// TIA Portal V16 export
// export: Created 2022-03-04T10:51:32.4810181Z, ExportSetting WithDefaults, DisplayName Totally Integrated Automation Portal, DisplayVersion V16 Update 3, DisplayName TIA Portal Version Control Interface, DisplayVersion V16 Update 2, DisplayName TIA Portal Openness, DisplayVersion V16 Update 3, DisplayName STEP 7 Professional, DisplayVersion V16 Update 3, DisplayName STEP 7 Safety, DisplayVersion V16, DisplayName WinCC Professional, DisplayVersion V16 Update 3
VAR_GLOBAL   // PLC tag table "FC19512"
   SIM001_TRIGGER AT %M900.0 : Bool;   // Simulation Trigger Signal
   SIM001_OUTPUT AT %MD910 : Real;
   SIM001_INPUT AT %MD902 : Real;
END_VAR
